// TIA Portal V20 export
FUNCTION_BLOCK "LER_visionHistory"   // FB32828, LAD
// stored: Access Published, MemoryReserve 100, SetENOAutomatically false
   VAR_INPUT
      save : Bool;
      partData : "LER_typePartData";
   END_VAR
   VAR_IN_OUT
      historyData : "LER_typeVisionHistory";
   END_VAR
   VAR
      statTonTime { ExternalAccessible := 'False'; ExternalVisible := 'False'; ExternalWritable := 'False'} : Array[0..9] of TON_TIME;
      statDeleteData { ExternalAccessible := 'False'; ExternalVisible := 'False'; ExternalWritable := 'False'} : "LER_typeVisionHistory";
      statPulse { ExternalAccessible := 'False'; ExternalVisible := 'False'; ExternalWritable := 'False'} : Bool;
      statComplete { ExternalAccessible := 'False'; ExternalVisible := 'False'; ExternalWritable := 'False'} : Bool;
   END_VAR
   VAR_TEMP
      tempRetVal : Array[0..9] of Int;
   END_VAR
   VAR_TEMP   // added for the SCL form of the ladder/FBD networks
      _w1 : Bool;
   END_VAR
BEGIN

REGION Network 1
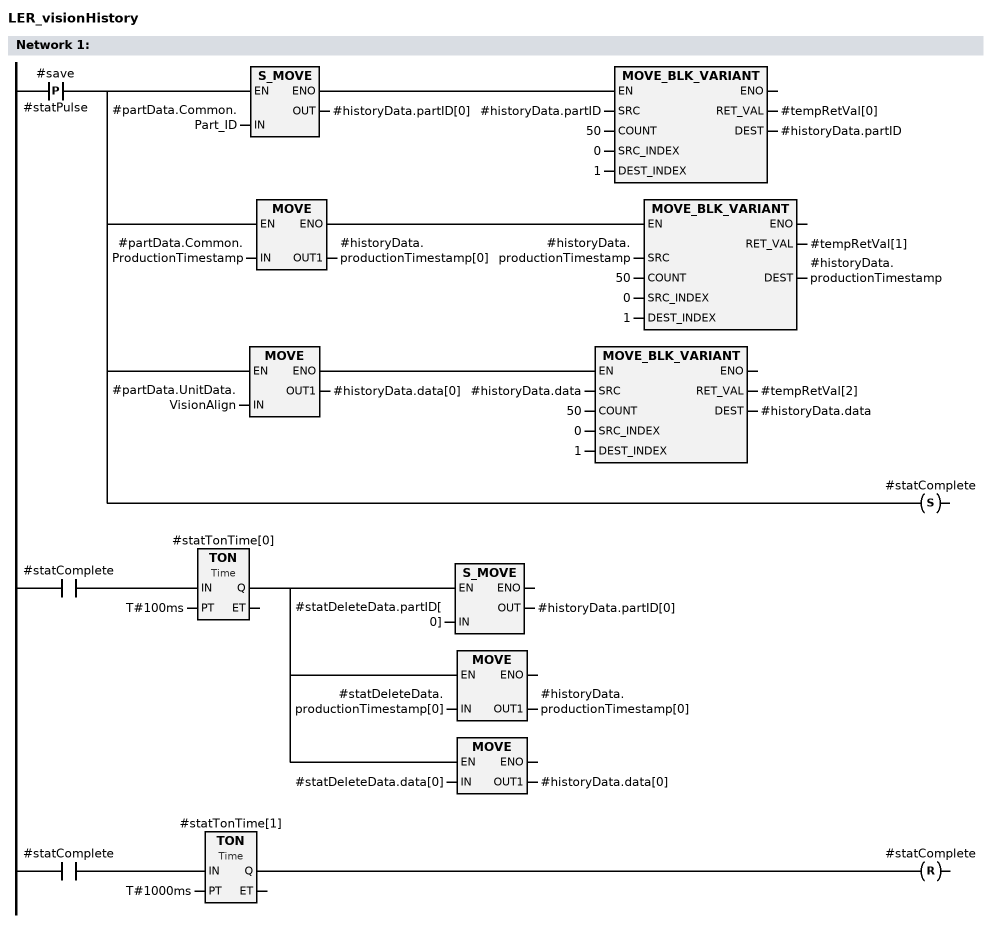
   RUNG wire#powerrail
      P_Contact(operand := #save, bit := #statPulse)
      wire#w1
      S_Move(in := #partData.Common.Part_ID, out => #historyData.partID[0])
      MOVE_BLK_VARIANT(SRC := #historyData.partID, COUNT := 50, SRC_INDEX := 0, DEST_INDEX := 1, Ret_Val => #tempRetVal[0], DEST => #historyData.partID)
   END_RUNG
   RUNG wire#w1
      Move(in := #partData.Common.ProductionTimestamp, out1 => #historyData.productionTimestamp[0])
      MOVE_BLK_VARIANT(SRC := #historyData.productionTimestamp, COUNT := 50, SRC_INDEX := 0, DEST_INDEX := 1, Ret_Val => #tempRetVal[1], DEST => #historyData.productionTimestamp)
   END_RUNG
   RUNG wire#w1
      Move(in := #partData.UnitData.VisionAlign, out1 => #historyData.data[0])
      MOVE_BLK_VARIANT(SRC := #historyData.data, COUNT := 50, SRC_INDEX := 0, DEST_INDEX := 1, Ret_Val => #tempRetVal[2], DEST => #historyData.data)
   END_RUNG
   RUNG wire#w1
      S_Coil( #statComplete )
   END_RUNG
   RUNG wire#powerrail
      Contact( #statComplete )
      { S7_Templates := "time_type := Time" } #statTonTime[0].TON(pt := T#100ms, et =>)
      wire#w2
      S_Move(in := #statDeleteData.partID[0], out => #historyData.partID[0])
   END_RUNG
   RUNG wire#w2
      Move(in := #statDeleteData.productionTimestamp[0], out1 => #historyData.productionTimestamp[0])
   END_RUNG
   RUNG wire#w2
      Move(in := #statDeleteData.data[0], out1 => #historyData.data[0])
   END_RUNG
   RUNG wire#powerrail
      Contact( #statComplete )
      { S7_Templates := "time_type := Time" } #statTonTime[1].TON(pt := T#1000ms, et =>)
      R_Coil( #statComplete )
   END_RUNG
   // the same network as SCL:
   #_w1 := #save AND NOT #statPulse;   // rising edge of #save
   #statPulse := #save;
   IF #_w1 THEN
       #historyData.partID[0] := #partData.Common.Part_ID;
       #tempRetVal[0] := MOVE_BLK_VARIANT(SRC := #historyData.partID,
                               COUNT := 50,
                               SRC_INDEX := 0,
                               DEST_INDEX := 1,
                               DEST => #historyData.partID);
       #historyData.productionTimestamp[0] := #partData.Common.ProductionTimestamp;
       #tempRetVal[1] := MOVE_BLK_VARIANT(SRC := #historyData.productionTimestamp,
                               COUNT := 50,
                               SRC_INDEX := 0,
                               DEST_INDEX := 1,
                               DEST => #historyData.productionTimestamp);
       #historyData.data[0] := #partData.UnitData.VisionAlign;
       #tempRetVal[2] := MOVE_BLK_VARIANT(SRC := #historyData.data,
                               COUNT := 50,
                               SRC_INDEX := 0,
                               DEST_INDEX := 1,
                               DEST => #historyData.data);
       #statComplete := TRUE;
   END_IF;
   #statTonTime[0].TON(IN := #statComplete, PT := T#100ms);
   IF #statTonTime[0].Q THEN
       #historyData.partID[0] := #statDeleteData.partID[0];
       #historyData.productionTimestamp[0] := #statDeleteData.productionTimestamp[0];
       #historyData.data[0] := #statDeleteData.data[0];
   END_IF;
   #statTonTime[1].TON(IN := #statComplete, PT := T#1000ms);
   IF #statTonTime[1].Q THEN #statComplete := FALSE; END_IF;
END_REGION
END_FUNCTION_BLOCK
